		//permissives to charge
		IF Permissives_DB.ReadyToCharge = TRUE THEN 
			FOR i := 1 TO n BY 1 DO 
				//MCP_IO.Charger[i].voltageSP := (HMI_DB.TDKLoad[i].RequiredChargedV *1000);
				MCP_IO.Charger[i].voltageSP := (1000*HMI_DB.TDKLoad[i].RequiredChargedV);
			END_FOR
		END_IF
		
		//start charging runout timer
		ChargingRunOutTMR_TON (IN := TRUE, PT := (ChargeTime_DB.LongestChargeTime_PT + HMI_DB.RunOutTMR_PT), ET => ChargingRunOutTMR_ET);
		
		IF Trips_DB.ChargingTimerRunout = TRUE THEN 
			StartChargingBroadcast := FALSE; // reset the broadcast bit whne all chargers
			ChargeTimeFinished := FALSE; //reset chargetime done bit
			ChargingRunOutTMR_TON (IN := FALSE);
			FOR i := 1 TO n BY 1 DO 
				ChargeTime_DB.ChargingTimeElapse_TON[i] (IN := FALSE);							
			END_FOR
			
			eState := E_State.ABORT; 
		END_IF
		
		IF Permissives_DB.AllChargeRelayClosed = TRUE THEN
			//start broadcasting on charger timer
			StartChargingBroadcast := TRUE;
		END_IF;
		//start timer 
		IF StartChargingBroadcast = TRUE THEN 
			//start total charge time TIMER
			ChargeTime_DB.LongestChargeTime_TON (IN := TRUE, PT := ChargeTime_DB.LongestChargeTime_PT, ET => ChargeTime_DB.LongestChargeTime_ET);
			
			//mapping HMI Charger Voltage SP to MCP IO 
			FOR i := 1 TO n BY 1 DO
				MCP_IO.Charger[i].voltageSP := (HMI_DB.TDKLoad[i].RequiredChargedV * 1000);
				//MCP_IO.Charger[1].voltageSP := REAL_TO_DINT (Setpoints.TDKLoad[1].RequiredChargedV);
			END_FOR;
			
			// delay stagger starts here
			ChargeTime_DB.ChargerDelay_TON[1] (IN := TRUE, PT := ChargeTime_DB.ChargerDelay_PT[1], ET => ChargeTime_DB.ChargerDelay_ET[1]);
			ChargeTime_DB.ChargerDelay_TON[2] (IN := TRUE, PT := ChargeTime_DB.ChargerDelay_PT[2], ET => ChargeTime_DB.ChargerDelay_ET[2]);
			ChargeTime_DB.ChargerDelay_TON[3] (IN := TRUE, PT := ChargeTime_DB.ChargerDelay_PT[3], ET => ChargeTime_DB.ChargerDelay_ET[3]);
		
			ChargeTime_DB.ChargerDelay_TON[4] (IN := TRUE, PT := ChargeTime_DB.ChargerDelay_PT[4], ET => ChargeTime_DB.ChargerDelay_ET[4]);
			ChargeTime_DB.ChargerDelay_TON[5] (IN := TRUE, PT := ChargeTime_DB.ChargerDelay_PT[5], ET => ChargeTime_DB.ChargerDelay_ET[5]);
			ChargeTime_DB.ChargerDelay_TON[6] (IN := TRUE, PT := ChargeTime_DB.ChargerDelay_PT[6], ET => ChargeTime_DB.ChargerDelay_ET[6]);
			//add shaft ramp
			ChargeTime_DB.ChargerDelay_TON[7] (IN := TRUE, PT := ChargeTime_DB.ChargerDelay_PT[7], ET => ChargeTime_DB.ChargerDelay_ET[7]);
			
			ELSE
				//Turn inhibit High on all chargers and turn off all timer if no broadcasting
				FOR i := 1 TO n BY 1 DO 
					MCP_IO.Charger[i].inhibit := TRUE; 
					MCP_IO.Charger[i].HV_ON := FALSE;
					// turn off timer
					ChargeTime_DB.ChargerDelay_TON[i] (IN := FALSE, PT := ChargeTime_DB.ChargerDelay_PT[i], ET => ChargeTime_DB.ChargerDelay_ET[i]);
				END_FOR;
		END_IF;
			
		FOR i := 1 TO n BY 1 DO	
			//turn on HV output to load	
			IF ChargeTime_DB.ChargerDelay_TON[i].Q = TRUE THEN
				StartCharger[i] := TRUE;
			END_IF	
			
			IF StartCharger[i] = TRUE (*AND Permissives.ReadyToCharge = TRUE*) THEN
				MCP_IO.Charger[i].HV_ON := TRUE;
				MCP_IO.Charger[i].inhibit := FALSE;
				ChargeTime_DB.ChargerDelay_TON[i] (IN := FALSE, PT := ChargeTime_DB.ChargerDelay_PT[i], ET => ChargeTime_DB.ChargerDelay_ET[i]);
				ChargeTime_DB.ChargingTimeElapse_TON[i]  (IN := TRUE, PT := REAL_TO_TIME (1000*MCP_IO.Charger[i].ChargeTime.timeToChargeLoad)); 
			END_IF;
			
			IF ChargeTime_DB.ChargingTimeElapse_TON[i].Q THEN
				StartCharger[i] := FALSE;
				ChargeTime_DB.ChargingTimeElapse_TON[i] (IN := FALSE); 
				//ChargeTime_DB.ChargerDelay_TON[i] (IN := FALSE, PT := ChargeTime_DB.ChargerDelay_PT[i], ET => ChargeTime_DB.ChargerDelay_ET[i]);
			END_IF;
		END_FOR;
				
		IF ChargingRunOutTMR_TON.Q = TRUE THEN
			Trips_DB.ChargingTimerRunout := TRUE;
			ChargingRunOutTMR_TON (IN := FALSE);
		END_IF;
		
		IF ChargeTime_DB.LongestChargeTime_TON.Q = TRUE THEN 
			ChargeTimeFinished := TRUE;
			StartChargingBroadcast := FALSE;
		
			ChargeTime_DB.LongestChargeTime_TON (IN := FALSE); //reset timer
		END_IF
		
		IF ChargeTimeFinished = TRUE THEN 
			
			FOR i := 1 TO n BY 1 DO 
				StartCharger[i] := FALSE;
				ChargeTime_DB.ChargingTimeElapse_TON[i] (IN := FALSE);							
			END_FOR
		END_IF
		
		//condition for charge complete
		IF Permissives_DB.AllChargerEOC = TRUE AND ChargeTimeFinished = TRUE (*all voltage reached*) THEN 
			ChargeCompleted := TRUE;
		//ELSE
			//ChargeCompleted := FALSE;
		END_IF
		
//if cap voltage feedback >= charger setpoints && EOC && all timer runout then chargecomplete
		IF ChargeCompleted = TRUE THEN 
			FOR i := 1 TO n BY 1 DO 
				MCP_IO.Charger[i].HV_ON := FALSE; 
				MCP_IO.Charger[i].inhibit := TRUE;
				
				StartCharger[i] := FALSE;
				ChargeTime_DB.ChargingTimeElapse_TON[i] (IN := FALSE);	
			END_FOR;
			ChargeRlyDelayON_Timer ( IN := TRUE, PT := ChargeRlyDelayON_PT);
		END_IF;

		IF ChargeRlyDelayON_Timer.Q = TRUE THEN
			ChargeRlyDelayDONE := TRUE;
		END_IF;

		IF ChargeRlyDelayDONE = TRUE THEN 	
			//Open all relays
			LCP1_IO.Segment[1].CloseChargeRly := FALSE;
			LCP1_IO.Segment[2].CloseChargeRly := FALSE;
			LCP1_IO.Segment[3].CloseChargeRly := FALSE;
				
			LCP2_IO.Segment[4].CloseChargeRly := FALSE;
			LCP2_IO.Segment[5].CloseChargeRly := FALSE;
			LCP2_IO.Segment[6].CloseChargeRly := FALSE;	
			
			//Shaft ramp
			LCP3_IO.CloseSRChargeRly := FALSE;
			
			//stagger the output - probably don't need to recheck this
//			LCP1_IO.Segment[1].OpenModule1To3DumpRly := TRUE;
//			LCP1_IO.Segment[2].OpenModule4To6DumpRly := TRUE;
//			LCP1_IO.Segment[3].OpenModule7To9DumpRly := TRUE;
//			LCP2_IO.Segment[4].OpenModule1To3DumpRly := TRUE;
//			LCP2_IO.Segment[5].OpenModule4To6DumpRly := TRUE;
//			LCP2_IO.Segment[6].OpenModule7To9DumpRly := TRUE;
			//shaft ramp - also does not need to recheck
			
			ChargeRlyDelayON_Timer ( IN := FALSE, PT := ChargeRlyDelayON_PT);							
			StartChargingBroadcast := FALSE; // reset the broadcast bit whne all chargers 
			
			eState := E_State.CHARGECOMPLETE;
		END_IF
		
	
	E_State.CHARGECOMPLETE:
		//keep led light on
		LCP1_IO.SegmentCharged := TRUE;
		LCP2_IO.SegmentCharged := TRUE;
		LCP3_IO.SegmentCharged := TRUE;
		
		ChargeRlyDelayDONE := FALSE;
		ChargeCompleted := FALSE;
		StartChargingBroadcast := FALSE; // reset the broadcast bit whne all chargers 
		ChargedRunOutTMR_TON (IN := TRUE, PT := HMI_DB.RunOutTMR_PT);
		ChargeRlyDelayON_Timer ( IN := FALSE, PT := ChargeRlyDelayON_PT);
		
		IF HMI_DB.FirePB = TRUE THEN 
			//LCP1_IO.Segment[1].Module[1].Fire := TRUE;
			LCP1_IO.TriggerScope := TRUE;
			LCP2_IO.TriggerScope := TRUE;
			ChargedRunOutTMR_TON (IN := FALSE);
			//and all other shot triggers.
			FirePBpressed := TRUE;
			//ELSE
				//LCP1_IO.Segment[1].Module[1].Fire := FALSE;
		END_IF
		
		IF FirePBpressed = TRUE THEN 
			//FireToSafeDelayTMR_TON (IN := TRUE, PT := FireToSafeDelayTMR_PT, ET => FireToSafeDelayTMR_ET);
			ShotTrigDelayTMR_TON (IN := TRUE, PT := ShotTrigDelayTMR_PT, ET => ShotTrigDelayTMR_ET);
			ScopeTrigPulseTMR_TON (IN := TRUE, PT := ScopeTrigPulseTMR_PT, ET => ScopeTrigPulseTMR_ET);
			ShotTrigPulseTMR_TON (IN := TRUE, PT := ShotTrigPulseTMR_PT, ET => ShotTrigPulseTMR_ET);
			//LCP1_IO.Segment[1].Module[1].Fire := TRUE;
		END_IF
		
		IF ScopeTrigPulseTMR_TON.Q = TRUE THEN 
			LCP1_IO.TriggerScope := FALSE;
			LCP2_IO.TriggerScope := FALSE;
			//ScopeTrigPulseTMR_TON (IN := FALSE);
		END_IF
		
		IF ShotTrigDelayTMR_TON.Q = TRUE THEN
			LCP1_IO.Fire := TRUE;
			LCP2_IO.Fire := TRUE;
			ShotFired := TRUE;
			//ShotTrigDelayTMR_TON (IN := FALSE);
		END_IF
		//might need to be a nested elsif
		IF ShotTrigPulseTMR_TON.Q = TRUE THEN
			LCP1_IO.Fire := FALSE;
			LCP2_IO.Fire := FALSE;
			//ShotTrigPulseTMR_TON (IN := FALSE);
		END_IF
		
		IF ShotFired = TRUE THEN
			FireToSafeDelayTMR_TON (IN := TRUE, PT := FireToSafeDelayTMR_PT, ET => FireToSafeDelayTMR_ET);
		END_IF
		
		IF FireToSafeDelayTMR_TON.Q = TRUE THEN
			FirePBpressed := FALSE;
			ShotFired := FALSE;
			FireToSafeDelayTMR_TON (IN := FALSE);
			ScopeTrigPulseTMR_TON (IN := FALSE);
			ShotTrigDelayTMR_TON (IN := FALSE);
			ShotTrigPulseTMR_TON (IN := FALSE);
			//LCP1_IO.Segment[1].Module[1].TriggerScope := FALSE;
			eState := E_State.SAFE;
		END_IF;
		
		IF ChargedRunOutTMR_TON.Q = TRUE THEN
			Trips_DB.ChargedTimerRunout := TRUE;
			ChargeTimeFinished := FALSE; //reset chargetime done bit
			ChargedRunOutTMR_TON (IN := FALSE);
			ScopeTrigPulseTMR_TON (IN := FALSE);
			ShotTrigDelayTMR_TON (IN := FALSE);
			ShotTrigPulseTMR_TON (IN := FALSE);
			eState := E_State.ABORT;
		END_IF

	E_State.DUMPING:

		// dump all 
		CompDumpStagger (start := FALSE, n := 6, reset := TRUE);
		LCP1_IO.Segment[1].OpenModule1To3DumpRly := FALSE;
		LCP1_IO.Segment[2].OpenModule4To6DumpRly := FALSE;
		LCP1_IO.Segment[3].OpenModule7To9DumpRly := FALSE;
		LCP2_IO.Segment[4].OpenModule1To3DumpRly := FALSE;
		LCP2_IO.Segment[5].OpenModule4To6DumpRly := FALSE;
		LCP2_IO.Segment[6].OpenModule7To9DumpRly := FALSE;
		
		SRDumpStagger (start := FALSE, n := 8, reset := TRUE);
		LCP3_IO.OpenSRDumpRly[1] := FALSE;
		LCP3_IO.OpenSRDumpRly[2] := FALSE;
		LCP3_IO.OpenSRDumpRly[3] := FALSE;
		LCP3_IO.OpenSRDumpRly[4] := FALSE;
		LCP3_IO.OpenSRDumpRly[5] := FALSE;
		LCP3_IO.OpenSRDumpRly[6] := FALSE;
		LCP3_IO.OpenSRDumpRly[7] := FALSE;
		LCP3_IO.OpenSRDumpRly[8] := FALSE;
		
		
		FOR i := 1 TO n BY 1 DO 
			MCP_IO.Charger[i].voltageSP := 0.001;
			MCP_IO.Charger[i].inhibit := TRUE;
			MCP_IO.Charger[i].HV_ON := FALSE;
		END_FOR;
		
		LCP1_IO.Segment[1].CloseChargeRly := FALSE;
		LCP1_IO.Segment[2].CloseChargeRly := FALSE;
		LCP1_IO.Segment[3].CloseChargeRly := FALSE;
		
		LCP2_IO.Segment[4].CloseChargeRly := FALSE;
		LCP2_IO.Segment[5].CloseChargeRly := FALSE;
		LCP2_IO.Segment[6].CloseChargeRly := FALSE;
		
		ChargeDelayStart := FALSE;
		FirePBpressed := FALSE;
		StartCharWarningTMR_TON (IN := FALSE, PT := StartCharWarningTMR_PT, ET=> StartCharWarningTMR_ET);
				
		DumpingRunOutTMR_TON (IN := TRUE, PT := DumpingRunOutTMR_PT);
		
		//HMI_DB.CloseChargeRlySW := FALSE;
		//HMI_DB.OpenDumpRlySW := FALSE;
		
		IF DumpingRunOutTMR_TON.Q = TRUE AND Permissives_DB.AllCapsDischarged = TRUE THEN
			eState := E_State.SAFE;
		END_IF

	E_State.ABORT:
		//dump all
		FOR i := 1 TO n BY 1 DO
			MCP_IO.Charger[i].inhibit := TRUE;
			MCP_IO.Charger[i].HV_ON := FALSE;
			MCP_IO.Charger[i].voltageSP := 0.001;
		END_FOR
				
		LCP1_IO.Segment[1].CloseChargeRly := FALSE;
		LCP1_IO.Segment[2].CloseChargeRly := FALSE;
		LCP1_IO.Segment[3].CloseChargeRly := FALSE;
		
		LCP2_IO.Segment[4].CloseChargeRly := FALSE;
		LCP2_IO.Segment[5].CloseChargeRly := FALSE;
		LCP2_IO.Segment[6].CloseChargeRly := FALSE;
		
		//reset stagger fg 
		CompDumpStagger (start := FALSE, n := 6, reset := TRUE);
		LCP1_IO.Segment[1].OpenModule1To3DumpRly := FALSE;
		LCP1_IO.Segment[2].OpenModule4To6DumpRly := FALSE;
		LCP1_IO.Segment[3].OpenModule7To9DumpRly := FALSE;
		LCP2_IO.Segment[4].OpenModule1To3DumpRly := FALSE;
		LCP2_IO.Segment[5].OpenModule4To6DumpRly := FALSE;
		LCP2_IO.Segment[6].OpenModule7To9DumpRly := FALSE;
		
		SRDumpStagger (start := FALSE, n := 6, reset := TRUE);
		LCP3_IO.OpenSRDumpRly[1] := FALSE;
		LCP3_IO.OpenSRDumpRly[2] := FALSE;
		LCP3_IO.OpenSRDumpRly[3] := FALSE;
		LCP3_IO.OpenSRDumpRly[4] := FALSE;
		LCP3_IO.OpenSRDumpRly[5] := FALSE;
		LCP3_IO.OpenSRDumpRly[6] := FALSE;
		LCP3_IO.OpenSRDumpRly[7] := FALSE;
		LCP3_IO.OpenSRDumpRly[8] := FALSE;
		
		HMI_DB.CloseChargeRlySW := FALSE;
		HMI_DB.OpenDumpRlySW := FALSE;
		HMI_DB.TurnChrgHVonSW := FALSE;
		HMI_DB.TurnChrgInhibitOffSW := FALSE;
		HMI_DB.TurnOnShotTrigSW := FALSE;
		HMI_DB.TurnOnChargeAlarm := FALSE;
		
		LCP1_IO.Fire := FALSE;
		LCP2_IO.Fire := FALSE;
		
		StartCharWarningTMR_TON (IN := FALSE);
		ChargeDelayStart := FALSE;
		FirePBpressed := FALSE;
	
		IF Permissives_DB.SystemIsSafe = TRUE AND Trips_DB.TimerRunOutON = FALSE THEN
			eState := E_State.SAFE;
		END_IF
		
	E_State.ManualMode:
		
		DumpingRunOutTMR_TON (IN := FALSE);
		StartCharWarningTMR_TON (IN := FALSE); // note
		
		LCP1_IO.Segment[1].CloseChargeRly := LCP1_IO.Segment[2].CloseChargeRly := LCP1_IO.Segment[3].CloseChargeRly := HMI_DB.CloseChargeRlySW;
		LCP2_IO.Segment[4].CloseChargeRly := LCP2_IO.Segment[5].CloseChargeRly := LCP2_IO.Segment[6].CloseChargeRly := HMI_DB.CloseChargeRlySW;
		LCP1_IO.Segment[1].OpenModule1To3DumpRly := LCP1_IO.Segment[2].OpenModule4To6DumpRly := LCP1_IO.Segment[3].OpenModule7To9DumpRly := HMI_DB.OpenDumpRlySW;
		LCP2_IO.Segment[4].OpenModule1To3DumpRly := LCP2_IO.Segment[5].OpenModule4To6DumpRly := LCP2_IO.Segment[6].OpenModule7To9DumpRly := HMI_DB.OpenDumpRlySW;
		
		IF HMI_DB.TurnChrgHVonSW = TRUE THEN
			FOR i := 1 TO n BY 1 DO 
				MCP_IO.Charger[i].HV_ON := TRUE;
			END_FOR
			ELSE
				FOR i := 1 TO n BY 1 DO 
					MCP_IO.Charger[i].HV_ON := FALSE;
				END_FOR
		END_IF
		
		IF HMI_DB.TurnChrgInhibitOffSW = TRUE THEN 
			FOR i := 1 TO n BY 1 DO 
				MCP_IO.Charger[i].inhibit := FALSE;
			END_FOR
			ELSE
				FOR i := 1 TO n BY 1 DO 
					MCP_IO.Charger[i].inhibit := TRUE;
				END_FOR				
		END_IF
		
		LCP1_IO.Fire := LCP2_IO.Fire := HMI_DB.TurnOnShotTrigSW;
		LCP1_IO.SegmentCharged := LCP2_IO.SegmentCharged := HMI_DB.TurnOnChargeAlarm;
		
		IF HMI_DB.HMI_ManualModeSelected = FALSE THEN
			eState := E_State.SAFE;
		END_IF
		
END_CASE;

IF i > n THEN 
	i := 1;
END_IF;	

IF j > 8 THEN 
	j := 1;
END_IF;	

IF k > 9 THEN 
	k := 1;
END_IF;	

IF m > 6 THEN 
	m := 4;
END_IF;

END_PROGRAM

// ---- POUs/Stagger_FB.TcPOU
FUNCTION_BLOCK Stagger_FB

VAR_INPUT
	start : BOOL := FALSE;
	n	  : INT := 8;
	reset : BOOL := FALSE;
END_VAR
VAR
	delayTMR_TON : TON;
	delayTMR_PT	 : TIME := T#100MS;
	delayTMR_ET	 : TIME;
	state		 : INT := 0;
	i			 : INT := 1;
	
	startOutput  : BOOL := 0;
END_VAR
VAR_OUTPUT
	OutputHi	: ARRAY[1..8] OF BOOL;

END_VAR

(* start goes high, stagger output sequence starts in a delay, 
	when the last output is high, it goes to idle,
	if reset goes high, it turns off all outputs - this fb needs to be reset when we dont want to output to be high.
	**to add, if both start and reset are high, throw a warning sign
*)
IF start = TRUE THEN 

CASE state OF
	0: 	//idle 	
//		FOR i := 1 TO n BY 1 DO 
//			OutputHi[i] := FALSE;
//		END_FOR
		delayTMR_TON (IN := FALSE, PT := delayTMR_PT, ET => delayTMR_ET);
		IF start = TRUE THEN 
			state := 1;
//			ELSIF reset = TRUE THEN 
//				state := 3;
//			ELSE 
//				state := 0;
		END_IF
		
	1: 	//output
		OutputHi[i] := TRUE;
		delayTMR_TON (IN := TRUE, PT := delayTMR_PT, ET => delayTMR_ET);
		
		IF delayTMR_TON.Q = TRUE THEN 
			state := 2;
		END_IF;
	2:	//increment
		delayTMR_TON (IN := FALSE, PT := delayTMR_PT, ET => delayTMR_ET);
		i := i + 1;
		
		IF OutputHi[n] = TRUE THEN 
			start := FALSE;
			state := 0;
		ELSE 
			IF i > n THEN 
				i := 1;
			END_IF
			state := 1;
		END_IF;
//	3:	//reset output 
//		FOR i := 1 TO n BY 1 DO 
//			OutputHi[i] := FALSE;
//		END_FOR
//		delayTMR_TON (IN := FALSE, PT := delayTMR_PT, ET => delayTMR_ET);
//		reset := 0; //debounce reset input
//		state := 0;
END_CASE

ELSIF reset = TRUE THEN 
		FOR i := 1 TO n BY 1 DO 
			OutputHi[i] := FALSE;
		END_FOR
		i := 1;
		state := 0;
END_IF;

IF i > n THEN 
	i := 1;
END_IF

END_FUNCTION_BLOCK

// ---- POUs/HMI.TcPOU
PROGRAM HMI
VAR
	eChargerType : E_ChargerType;
	
	SysCLK					: GETSYSTEMTIME;
	//fileTime				: T_FILETIME;
	LastTimeShot			: STRING;
	ChargeGraphTMR_TON		: TON;
	ChargeGraphTMR_PT		: TIME := ChargeTime_DB.LongestChargeTime_PT + T#10S;
	ChargeGraphTMR_ET		: TIME;
	LongestChargeTIME		: REAL;
	LastTimeShotLog			: BOOL;
	
	i : INT := 1;
	n : INT := 7;

	LastTimeShotTMR_TON		: TON;
	LastTimeShotTMR_PT		: TIME := T#120H;
	LastTimeShotTMR_ET		: TIME;
	LastTimeShotTMR_REAL	: DWORD;
END_VAR

// if clear all faults, reset abort status
IF HMI_DB.ClearFaultPB = TRUE THEN
	Trips_DB.ChargedTimerRunout := FALSE;
	Trips_DB.ChargingTimerRunout := FALSE;
	Trips_DB.DumpTimerRunout := FALSE;
	Trips_DB.ChargerSummaryFault := FALSE;
	Trips_DB.ShortingSystemUnknown := FALSE;
	Trips_DB.AnyEstopPressed := FALSE;
END_IF

IF Trips_DB.ChargedTimerRunout = TRUE OR 
	Trips_DB.ChargingTimerRunout = TRUE //OR 
	//Trips_DB.DumpTimerRunout = TRUE 
	THEN
		Trips_DB.TimerRunOutON := TRUE; 
		ELSE
			Trips_DB.TimerRunOutON := FALSE;
		END_IF
		
FOR i := 1 TO n BY 1 DO 
	MCP_IO.Charger[i].ChargerType := Setpoints.TDKLoad[i].eChargerType := HMI_DB.TDKLoad[i].eChargerType;
		
	IF MCP_IO.Charger[i].ChargerType = E_ChargerType.TDK12kV THEN 
		HMI_DB.TDKLoad[i].PSratedV := 12;
		ELSIF MCP_IO.Charger[i].ChargerType = E_ChargerType.TDK30kV THEN
			HMI_DB.TDKLoad[i].PSratedV := 30;
		ELSIF MCP_IO.Charger[i].ChargerType = E_ChargerType.TDK50kV THEN
			HMI_DB.TDKLoad[i].PSratedV := 50;
	END_IF
END_FOR;

LastTimeShotTMR_TON (IN := TRUE, PT := LastTimeShotTMR_PT, ET => LastTimeShotTMR_ET);

IF (Sequence.eState = E_State.CHARGECOMPLETE) AND HMI_DB.FirePB = TRUE THEN 
	//SysCLK (timeLoDW => fileTime.dwLowDateTime, timeHiDW => fileTime.dwHighDateTime);
	//LastTimeShot := SYSTEMTIME_TO_STRING( FILETIME_TO_SYSTEMTIME( fileTime ) );	
	LastTimeShotTMR_TON (IN := FALSE, PT := LastTimeShotTMR_PT, ET => LastTimeShotTMR_ET);
	HMI_DB.LastTimeShotLog := TRUE;	
	ELSE
		HMI_DB.LastTimeShotLog := FALSE;
END_IF

LastTimeShotTMR_REAL := TIME_TO_DWORD (LastTimeShotTMR_ET)/1000;

IF (Sequence.eState = E_State.CHARGECOMPLETE OR Sequence.eState = E_State.CHARGING) THEN
	ChargeGraphTMR_TON (IN:= TRUE, PT:= ChargeGraphTMR_PT, ET => ChargeGraphTMR_ET);
	ELSE
		ChargeGraphTMR_TON (IN:= FALSE);
END_IF

LongestChargeTIME := TIME_TO_REAL (ChargeGraphTMR_ET)/1000;

IF i > n THEN 
	i := 1;
END_IF

END_PROGRAM

// ---- POUs/Alarms.TcPOU
PROGRAM Alarms
VAR
	bWarning : BOOL;
	bConfirm : BOOL;
	alarms : ARRAY[0..32] OF Alarms_FB;
	
END_VAR

// Alarm Word 1 - MCP Alarms
//MCP Alarms

Alarms_DB.MCP.AlarmWord.0 := Trips_DB.AnyEstopPressed;
Alarms_DB.MCP.AlarmWord.1 := Trips_DB.CageDoorNotClose;
Alarms_DB.MCP.AlarmWord.2 := Trips_DB.ShortingSystemUnknown;
Alarms_DB.MCP.AlarmWord.3 := Trips_DB.MasterSTOPPressed;
Alarms_DB.MCP.AlarmWord.4 := MCP_IO.Charger[1].SummaryFaulted;
Alarms_DB.MCP.AlarmWord.5 := MCP_IO.Charger[2].SummaryFaulted;
Alarms_DB.MCP.AlarmWord.6 := MCP_IO.Charger[3].SummaryFaulted;
Alarms_DB.MCP.AlarmWord.7 := MCP_IO.Charger[4].SummaryFaulted;
Alarms_DB.MCP.AlarmWord.8 := MCP_IO.Charger[5].SummaryFaulted;
Alarms_DB.MCP.AlarmWord.9 := MCP_IO.Charger[6].SummaryFaulted;
//Alarms_DB.MCP.AlarmWord.10 := MCP_IO.Charger[7].SummaryFaulted;
Alarms_DB.MCP.AlarmWord.11 := Permissives_DB.AnyVoltMonBoardLoss;
Alarms_DB.MCP.AlarmWord.12 := Trips_DB.ChargedTimerRunout;
Alarms_DB.MCP.AlarmWord.13 := Trips_DB.ChargingTimerRunout;
Alarms_DB.MCP.AlarmWord.14 := HMI_DB.LastTimeShotLog;
//Alarms_DB.MCP.AlarmWord.15 := Trips_DB.AnyEstopPressed;

//Alarm Word 1 msg
//IE: alarms[299](evtEntry:= Tc_Events.AlarmWord11.b4, bEvt:= gvl.test, bConfirm:= bConfirm);
alarms[0](evtEntry:= Tc_Events.AlarmWord1.b0, bEvt:= Alarms_DB.MCP.AlarmWord.0, bConfirm:= bConfirm);
alarms[1](evtEntry:= Tc_Events.AlarmWord1.b1, bEvt:= Alarms_DB.MCP.AlarmWord.1, bConfirm:= bConfirm);
alarms[2](evtEntry:= Tc_Events.AlarmWord1.b2, bEvt:= Alarms_DB.MCP.AlarmWord.2, bConfirm:= bConfirm);
alarms[3](evtEntry:= Tc_Events.AlarmWord1.b3, bEvt:= Alarms_DB.MCP.AlarmWord.3, bConfirm:= bConfirm);
alarms[4](evtEntry:= Tc_Events.AlarmWord1.b4, bEvt:= Alarms_DB.MCP.AlarmWord.4, bConfirm:= bConfirm);
alarms[5](evtEntry:= Tc_Events.AlarmWord1.b5, bEvt:= Alarms_DB.MCP.AlarmWord.5, bConfirm:= bConfirm);
alarms[6](evtEntry:= Tc_Events.AlarmWord1.b6, bEvt:= Alarms_DB.MCP.AlarmWord.6, bConfirm:= bConfirm);
alarms[7](evtEntry:= Tc_Events.AlarmWord1.b7, bEvt:= Alarms_DB.MCP.AlarmWord.7, bConfirm:= bConfirm);
alarms[8](evtEntry:= Tc_Events.AlarmWord1.b8, bEvt:= Alarms_DB.MCP.AlarmWord.8, bConfirm:= bConfirm);
alarms[9](evtEntry:= Tc_Events.AlarmWord1.b9, bEvt:= Alarms_DB.MCP.AlarmWord.9, bConfirm:= bConfirm);
alarms[0](evtEntry:= Tc_Events.AlarmWord1.b10, bEvt:= Alarms_DB.MCP.AlarmWord.10, bConfirm:= bConfirm);
alarms[11](evtEntry:= Tc_Events.AlarmWord1.b11, bEvt:= Alarms_DB.MCP.AlarmWord.11, bConfirm:= bConfirm);
alarms[12](evtEntry:= Tc_Events.AlarmWord1.b12, bEvt:= Alarms_DB.MCP.AlarmWord.12, bConfirm:= bConfirm);
alarms[13](evtEntry:= Tc_Events.AlarmWord1.b13, bEvt:= Alarms_DB.MCP.AlarmWord.13, bConfirm:= bConfirm);
alarms[14](evtEntry:= Tc_Events.AlarmWord1.b14, bEvt:= Alarms_DB.MCP.AlarmWord.14, bConfirm:= bConfirm);
alarms[15](evtEntry:= Tc_Events.AlarmWord1.b15, bEvt:= Alarms_DB.MCP.AlarmWord.15, bConfirm:= bConfirm);

// Alarm Word 2 - Section 1 Alarms
(*Alarms_DB.Section1.AlarmWord.0 := Trips_DB.Section[1].SystemTripped;
Alarms_DB.Section1.AlarmWord.1 := Trips_DB.Section[1].LossPneumaticPressure;
Alarms_DB.Section1.AlarmWord.2 := Trips_DB.Section[1].Peak.ChargeRelay1_Failed;
Alarms_DB.Section1.AlarmWord.3 := Trips_DB.Section[1].Peak.ChargeRelay2_Failed;
Alarms_DB.Section1.AlarmWord.4 := Trips_DB.Section[1].Peak.DumpRelay1_Failed;
Alarms_DB.Section1.AlarmWord.5 := Trips_DB.Section[1].Peak.DumpRelay2_Failed;
Alarms_DB.Section1.AlarmWord.6 := Trips_DB.Section[1].Sust.ChargeRelay1_Failed;
Alarms_DB.Section1.AlarmWord.7 := Trips_DB.Section[1].Sust.ChargeRelay2_Failed;
Alarms_DB.Section1.AlarmWord.8 := Trips_DB.Section[1].Sust.DumpRelay1_Failed;
Alarms_DB.Section1.AlarmWord.9 := Trips_DB.Section[1].Sust.DumpRelay2_Failed;
Alarms_DB.Section1.AlarmWord.10 := Trips_DB.Section[1].LossDCPower;


// Alarm Word 2 - Msg
alarms[16](evtEntry:= Tc_Events.AlarmWord2.b0, bEvt:= Alarms_DB.Section1.AlarmWord.0, bConfirm:= bConfirm);
alarms[17](evtEntry:= Tc_Events.AlarmWord2.b1, bEvt:= Alarms_DB.Section1.AlarmWord.1, bConfirm:= bConfirm);
alarms[18](evtEntry:= Tc_Events.AlarmWord2.b2, bEvt:= Alarms_DB.Section1.AlarmWord.2, bConfirm:= bConfirm);
alarms[19](evtEntry:= Tc_Events.AlarmWord2.b3, bEvt:= Alarms_DB.Section1.AlarmWord.3, bConfirm:= bConfirm);
alarms[20](evtEntry:= Tc_Events.AlarmWord2.b4, bEvt:= Alarms_DB.Section1.AlarmWord.4, bConfirm:= bConfirm);
alarms[21](evtEntry:= Tc_Events.AlarmWord2.b5, bEvt:= Alarms_DB.Section1.AlarmWord.5, bConfirm:= bConfirm);
alarms[22](evtEntry:= Tc_Events.AlarmWord2.b6, bEvt:= Alarms_DB.Section1.AlarmWord.6, bConfirm:= bConfirm);
alarms[23](evtEntry:= Tc_Events.AlarmWord2.b7, bEvt:= Alarms_DB.Section1.AlarmWord.7, bConfirm:= bConfirm);
alarms[24](evtEntry:= Tc_Events.AlarmWord2.b8, bEvt:= Alarms_DB.Section1.AlarmWord.8, bConfirm:= bConfirm);
alarms[25](evtEntry:= Tc_Events.AlarmWord2.b9, bEvt:= Alarms_DB.Section1.AlarmWord.9, bConfirm:= bConfirm);
alarms[26](evtEntry:= Tc_Events.AlarmWord2.b10, bEvt:= Alarms_DB.Section1.AlarmWord.10, bConfirm:= bConfirm);
//alarms[27] - spare
//alarms[28] - spare
//alarms[29] - spare
//alarms[30] - spare
//alarms[31] - spare
*)

//Clear Alarm Word
IF bConfirm THEN
	Alarms_DB.MCP.AlarmWord := 0;
	Alarms_DB.Segment1.AlarmWord := 0;
	
	(*Alarms_DB.Coil3.AlarmWord := 0;
	Alarms_DB.Coil4.AlarmWord := 0;
	Alarms_DB.Coil5.AlarmWord := 0;
	Alarms_DB.Coil6.AlarmWord := 0;
	Alarms_DB.Coil7.AlarmWord := 0;
	Alarms_DB.Coil8.AlarmWord := 0;
	Alarms_DB.Coil9.AlarmWord := 0;
	Alarms_DB.Coil10.AlarmWord := 0;
	Alarms_DB.AlarmWord_11.AlarmWord := 0;
	Alarms_DB.AlarmWord_22.AlarmWord := 0;
	Alarms_DB.AlarmWord_23.AlarmWord := 0;
	Alarms_DB.AlarmWord_24.AlarmWord := 0;
	Alarms_DB.AlarmWord_25.AlarmWord := 0;
	Alarms_DB.AlarmWord_26.AlarmWord := 0;
	Alarms_DB.AlarmWord_27.AlarmWord := 0;
	*)
END_IF;

END_PROGRAM

// ---- POUs/Alarms_FB.TcPOU
FUNCTION_BLOCK Alarms_FB EXTENDS FB_TcAlarm
VAR_INPUT
	evtEntry : TcEventEntry;
	bEvt : BOOL;
	bConfirm : BOOL;
END_VAR
VAR_OUTPUT
END_VAR
VAR
	bInit  : BOOL := TRUE;
	bMem : BOOL;
END_VAR

IF bInit THEN
	SUPER^.CreateEx(evtEntry, TRUE, 0);
	bInit := FALSE;
END_IF

IF bEvt AND NOT bMem AND SUPER^.eConfirmationState <> TcEventConfirmationState.WaitForConfirmation THEN
	SUPER^.Raise(0);
END_IF

IF bMem AND NOT bEvt THEN
	SUPER^.Clear(0, FALSE);
END_IF

IF bConfirm THEN
	SUPER^.Confirm(0);
END_IF
bMem := bEvt;

END_FUNCTION_BLOCK
